(* CODESYS project TrafficLight-skeleton.project

Project tree, tasks and I/O mapping:
  Device : CODESYS Control Win V3, 3S - Smart Software Solutions GmbH, version 3.5.15.30
    application Application
      libraries: Standard, * (System)
      task MainTask (cyclic, interval t#20ms, priority 1) calls PLC_PRG
      program PLC_PRG [FBD]
      function block NormalCycle_FB [ST]
      function block BlinkingYellow_FB [ST]
*)

// Device/Application/PLC_PRG
PROGRAM PLC_PRG
VAR
	TON_0: TON;
	Normal_FSM: NormalCycle_FB;
	Blinking_FSM: BlinkingYellow_FB;
END_VAR

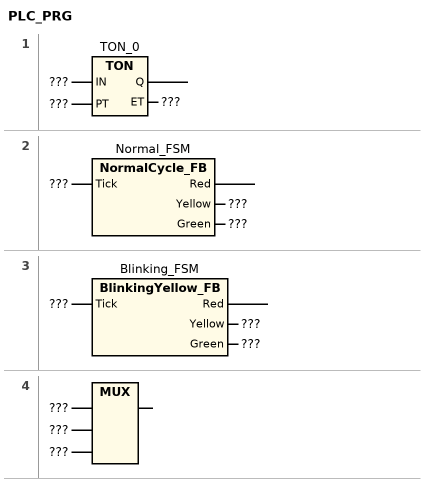
// NETWORK 1
TON_0(); // TON

// NETWORK 2
Normal_FSM(); // NormalCycle_FB

// NETWORK 3
Blinking_FSM(); // BlinkingYellow_FB

// NETWORK 4
MUX(???, ???, ???);

END_PROGRAM

// Device/Application/NormalCycle_FB
FUNCTION_BLOCK NormalCycle_FB
(* Add other vars here *)
VAR_INPUT
	Tick : BOOL;
END_VAR
VAR_OUTPUT
	Red : BOOL;
	Yellow : BOOL;
	Green : BOOL;
	
END_VAR
VAR
	State : WORD;
	Counter : WORD;
END_VAR

(* Add your logics here *)

END_FUNCTION_BLOCK

// Device/Application/BlinkingYellow_FB
FUNCTION_BLOCK BlinkingYellow_FB
(* Add other vars here *)
VAR_INPUT
	Tick : BOOL;
END_VAR
VAR_OUTPUT
	Red : BOOL;
	Yellow : BOOL;
	Green : BOOL;
END_VAR
VAR
	State : WORD;
END_VAR

(* Add your logics here *)

END_FUNCTION_BLOCK
